TYPE ProcessDataObjectIndex : STRUCT
    index : WORD;
    subIndex : BYTE;
END_STRUCT
END_TYPE

(* stored: Version 1.1.0.1
   DUT ProcessDataObjectIndex: Id {72581df7-23a1-0c07-10c2-55288759defe} *)
